
// ===== library: MasterCopy "Pallet dispenser" =====

FUNCTION_BLOCK "Pallet dispenser"   // FB4, LAD
{ S7_Optimized_Access := 'FALSE' }
VERSION : 0.1
   VAR_INPUT
      DOWN_accident : Bool;
      Dispenser_is_down : Bool;
      Dispenser_in_middle : Bool;
      Dispenser_is_up : Bool;
      UP_accident : Bool;
      Circuit_breaker : Bool;
      Arms_are_open : Bool;
      Arms_are_close : Bool;
      Pallet_under_dispenser : Bool;
      Automatic_mode : Bool;
      Power_circuit_OK : Bool;
      Pneumatic_OK : Bool;
      Sensor_before_dispenser : Bool;
      Button_Open_door : Bool;
      Sensor_door_are_open : Bool;
      Button_Door_are_close : Bool;
      OP_up : Bool;
      OP_down : Bool;
      OP_Airs_move : Bool;
      Pallet_transfare : Bool;
      Button_RESET : Bool;
   END_VAR
   VAR_OUTPUT
      Let_go_UP : Bool;
      Let_go_DOWN : Bool;
      Break : Bool;
      Let_arms_close : Bool;
      Let_arms_open : Bool;
      Let_open_door : Bool;
      Led_door_are_open : Bool;
   END_VAR
   VAR
      Paleta_polozena : Bool;
      Stop_v_rucnim : Bool;
      Hrana_stop_v_rucnim : Bool;
      Pozadavek_otevreni_dveri : Bool;
      Door_opened : Bool;
      Arms_are_close_pozition : Bool;
   END_VAR
   VAR_TEMP   // added for the SCL form of the ladder/FBD networks
      _s5time1 : S5Time;
      _w1 : Bool;
   END_VAR
BEGIN

REGION Network 1
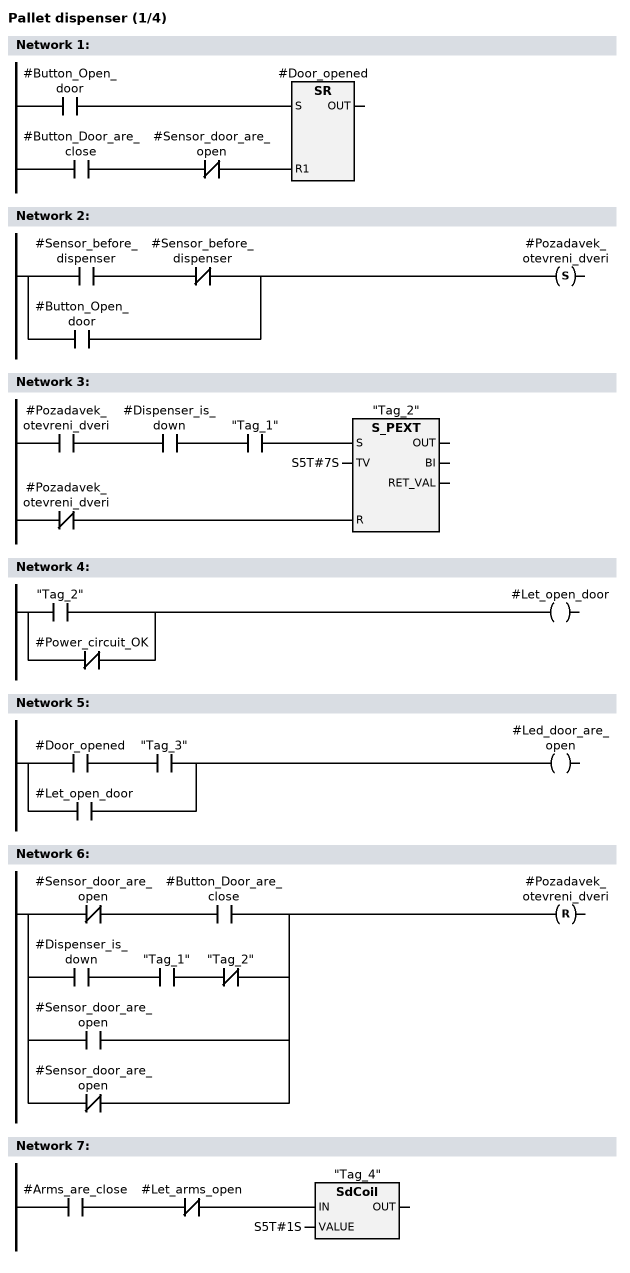
   IF #Button_Open_door THEN
       #Door_opened := TRUE;   // SR flip-flop
   END_IF;
   IF #Button_Door_are_close AND NOT #Sensor_door_are_open THEN #Door_opened := FALSE; END_IF;
END_REGION

REGION Network 2
   RUNG wire#powerrail
      Contact( #Sensor_before_dispenser )
      I_Contact( #Sensor_before_dispenser )
      wire#w1
      S_Coil( #Pozadavek_otevreni_dveri )
   END_RUNG
   RUNG wire#powerrail
      Contact( #Button_Open_door )
   END_RUNG wire#w1
   // the same network as SCL:
   IF (#Sensor_before_dispenser AND NOT #Sensor_before_dispenser) OR #Button_Open_door THEN
       #Pozadavek_otevreni_dveri := TRUE;
   END_IF;
END_REGION

REGION Network 3
   RUNG wire#powerrail
      Contact( #Pozadavek_otevreni_dveri )
      Contact( #Dispenser_is_down )
      Contact( "Tag_1" )
      S_PEXT(T_NO := "Tag_2", TV := S5T#7S, R := wire#w1, BI =>, RET_VAL =>)
   END_RUNG
   RUNG wire#powerrail
      I_Contact( #Pozadavek_otevreni_dveri )
   END_RUNG wire#w1
   // the same network as SCL:
   #_s5time1 := S_PEXT(T_NO := "Tag_2",
                       TV := S5T#7S,
                       S := #Pozadavek_otevreni_dveri AND #Dispenser_is_down AND "Tag_1",
                       R := NOT #Pozadavek_otevreni_dveri);
END_REGION

REGION Network 4
   RUNG wire#powerrail
      Contact( "Tag_2" )
      wire#w1
      Coil( #Let_open_door )
   END_RUNG
   RUNG wire#powerrail
      I_Contact( #Power_circuit_OK )
   END_RUNG wire#w1
   // the same network as SCL:
   #Let_open_door := "Tag_2" OR NOT #Power_circuit_OK;
END_REGION

REGION Network 5
   #Led_door_are_open := #Let_open_door OR (#Door_opened AND "Tag_3");
END_REGION

REGION Network 6
   RUNG wire#powerrail
      I_Contact( #Sensor_door_are_open )
      Contact( #Button_Door_are_close )
      wire#w1
      R_Coil( #Pozadavek_otevreni_dveri )
   END_RUNG
   RUNG wire#powerrail
      Contact( #Dispenser_is_down )
      Contact( "Tag_1" )
      I_Contact( "Tag_2" )
   END_RUNG wire#w1
   RUNG wire#powerrail
      Contact( #Sensor_door_are_open )
   END_RUNG wire#w1
   RUNG wire#powerrail
      I_Contact( #Sensor_door_are_open )
   END_RUNG wire#w1
   // the same network as SCL:
   IF (NOT #Sensor_door_are_open AND #Button_Door_are_close) OR (#Dispenser_is_down AND "Tag_1" AND NOT "Tag_2") OR #Sensor_door_are_open OR NOT #Sensor_door_are_open THEN
       #Pozadavek_otevreni_dveri := FALSE;
   END_IF;
END_REGION

REGION Network 7
   // no SCL statement known for SdCoil: written as a call
   SdCoil(value := S5T#1S, operand := "Tag_4", in := #Arms_are_close AND NOT #Let_arms_open);
END_REGION

REGION Network 8
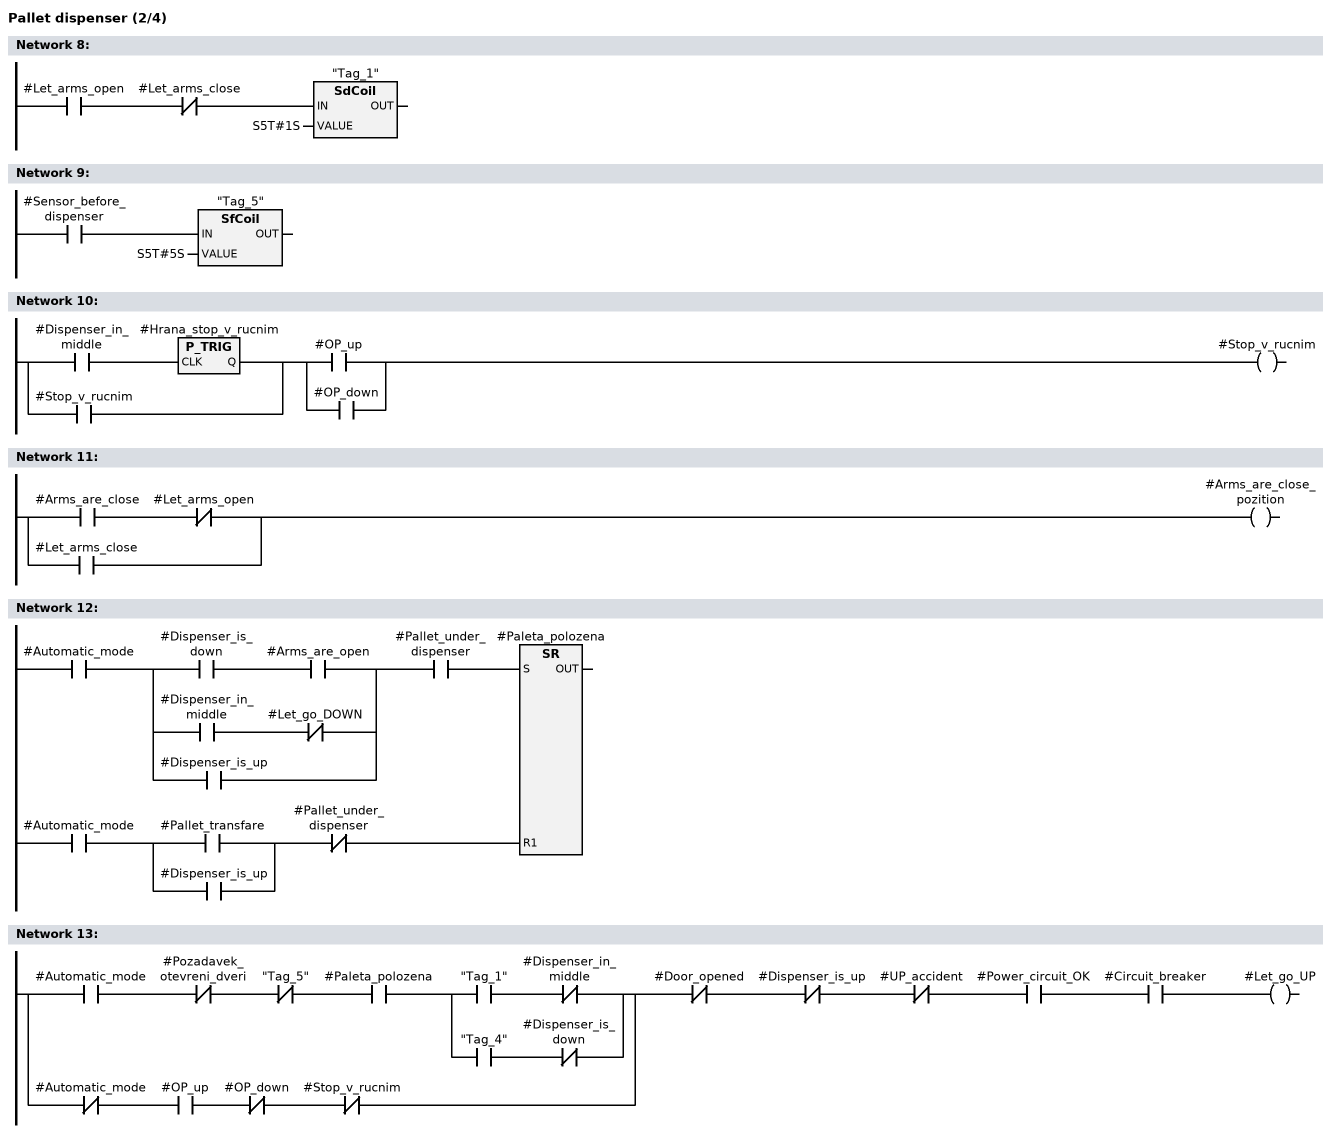
   // no SCL statement known for SdCoil: written as a call
   SdCoil(value := S5T#1S, operand := "Tag_1", in := #Let_arms_open AND NOT #Let_arms_close);
END_REGION

REGION Network 9
   // no SCL statement known for SfCoil: written as a call
   SfCoil(value := S5T#5S, operand := "Tag_5", in := #Sensor_before_dispenser);
END_REGION

REGION Network 10
   RUNG wire#powerrail
      Contact( #Dispenser_in_middle )
      P_Trig( #Hrana_stop_v_rucnim )
      wire#w1
      Contact( #OP_up )
      wire#w2
      Coil( #Stop_v_rucnim )
   END_RUNG
   RUNG wire#powerrail
      Contact( #Stop_v_rucnim )
   END_RUNG wire#w1
   RUNG wire#w1
      Contact( #OP_down )
   END_RUNG wire#w2
   // the same network as SCL:
   #_w1 := #Dispenser_in_middle AND NOT #Hrana_stop_v_rucnim;   // rising edge
   #Hrana_stop_v_rucnim := #Dispenser_in_middle;
   #Stop_v_rucnim := (#_w1 OR #Stop_v_rucnim) AND (#OP_up OR #OP_down);
END_REGION

REGION Network 11
   RUNG wire#powerrail
      Contact( #Arms_are_close )
      I_Contact( #Let_arms_open )
      wire#w1
      Coil( #Arms_are_close_pozition )
   END_RUNG
   RUNG wire#powerrail
      Contact( #Let_arms_close )
   END_RUNG wire#w1
   // the same network as SCL:
   #Arms_are_close_pozition := (#Arms_are_close AND NOT #Let_arms_open) OR #Let_arms_close;
END_REGION

REGION Network 12
   IF #Automatic_mode AND ((#Dispenser_is_down AND #Arms_are_open) OR (#Dispenser_in_middle AND NOT #Let_go_DOWN) OR #Dispenser_is_up) AND #Pallet_under_dispenser THEN
       #Paleta_polozena := TRUE;   // SR flip-flop
   END_IF;
   IF #Automatic_mode AND (#Pallet_transfare OR #Dispenser_is_up) AND NOT #Pallet_under_dispenser THEN
       #Paleta_polozena := FALSE;
   END_IF;
END_REGION

REGION Network 13
   #Let_go_UP := ((#Automatic_mode AND NOT #Pozadavek_otevreni_dveri AND NOT "Tag_5" AND #Paleta_polozena AND (("Tag_1" AND NOT #Dispenser_in_middle) OR ("Tag_4" AND NOT #Dispenser_is_down))) OR (NOT #Automatic_mode AND #OP_up AND NOT #OP_down AND NOT #Stop_v_rucnim)) AND NOT #Door_opened AND NOT #Dispenser_is_up AND NOT #UP_accident AND #Power_circuit_OK AND #Circuit_breaker;
END_REGION

REGION Network 14
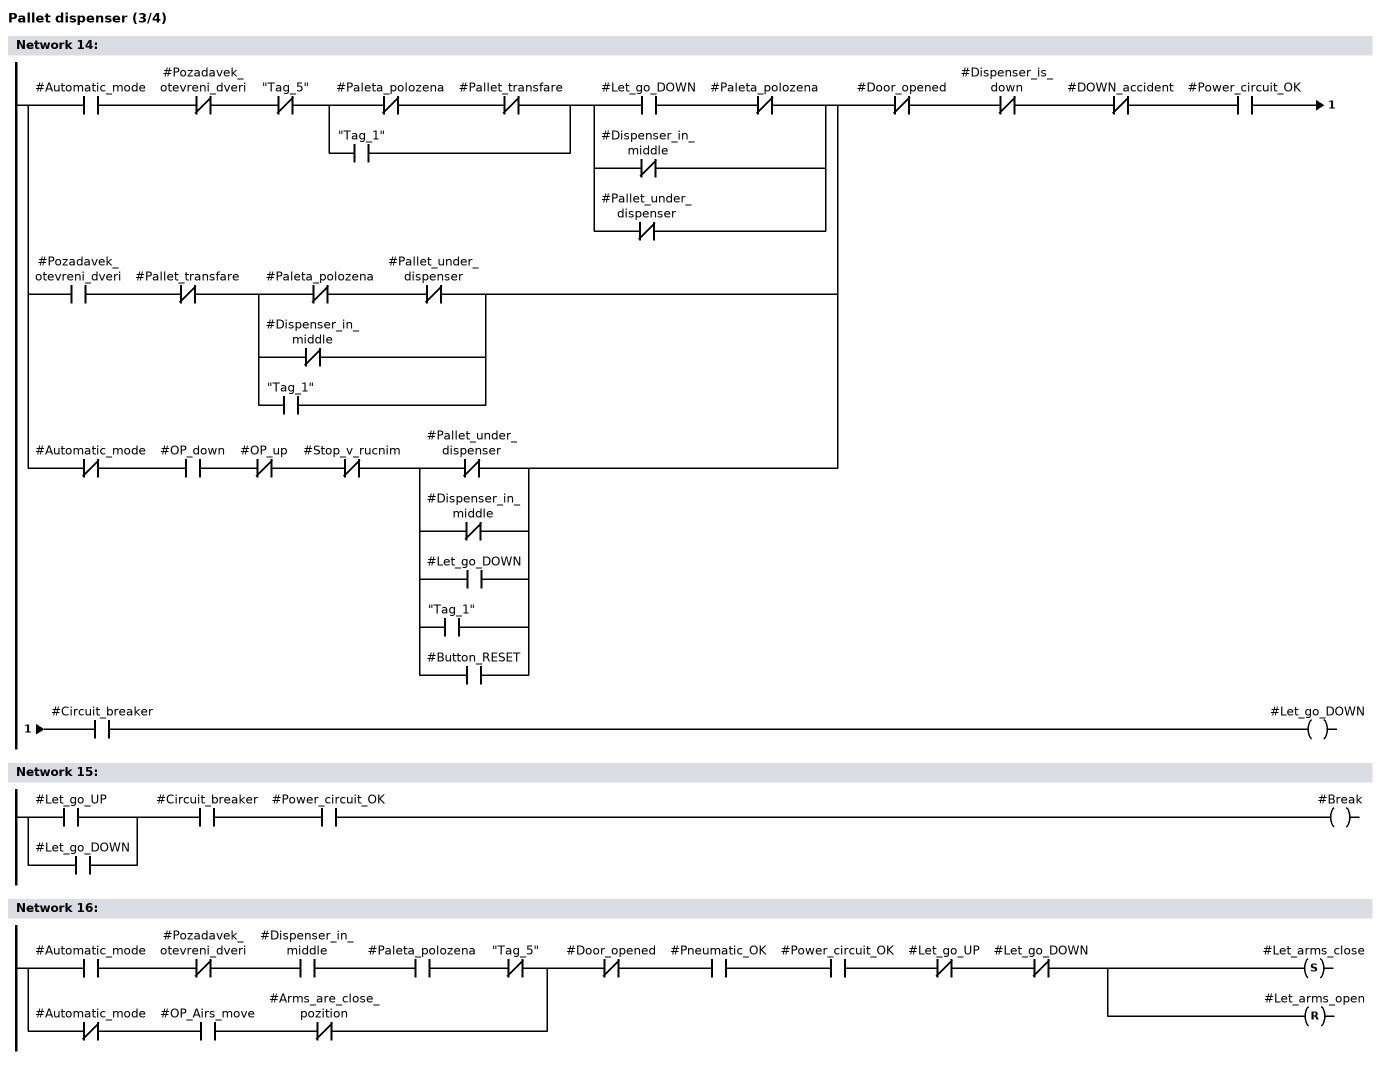
   #Let_go_DOWN := ((#Automatic_mode AND NOT #Pozadavek_otevreni_dveri AND NOT "Tag_5" AND ((NOT #Paleta_polozena AND NOT #Pallet_transfare) OR "Tag_1") AND (NOT #Dispenser_in_middle OR NOT #Pallet_under_dispenser OR (#Let_go_DOWN AND NOT #Paleta_polozena))) OR (#Pozadavek_otevreni_dveri AND NOT #Pallet_transfare AND (NOT #Dispenser_in_middle OR (NOT #Paleta_polozena AND NOT #Pallet_under_dispenser) OR "Tag_1")) OR (NOT #Automatic_mode AND #OP_down AND NOT #OP_up AND NOT #Stop_v_rucnim AND (NOT #Pallet_under_dispenser OR NOT #Dispenser_in_middle OR #Let_go_DOWN OR "Tag_1" OR #Button_RESET))) AND NOT #Door_opened AND NOT #Dispenser_is_down AND NOT #DOWN_accident AND #Power_circuit_OK AND #Circuit_breaker;
END_REGION

REGION Network 15
   RUNG wire#powerrail
      Contact( #Let_go_UP )
      wire#w1
      Contact( #Circuit_breaker )
      Contact( #Power_circuit_OK )
      Coil( #Break )
   END_RUNG
   RUNG wire#powerrail
      Contact( #Let_go_DOWN )
   END_RUNG wire#w1
   // the same network as SCL:
   #Break := (#Let_go_UP OR #Let_go_DOWN) AND #Circuit_breaker AND #Power_circuit_OK;
END_REGION

REGION Network 16
   RUNG wire#powerrail
      Contact( #Automatic_mode )
      I_Contact( #Pozadavek_otevreni_dveri )
      Contact( #Dispenser_in_middle )
      Contact( #Paleta_polozena )
      I_Contact( "Tag_5" )
      wire#w1
      I_Contact( #Door_opened )
      Contact( #Pneumatic_OK )
      Contact( #Power_circuit_OK )
      I_Contact( #Let_go_UP )
      I_Contact( #Let_go_DOWN )
      wire#w2
      S_Coil( #Let_arms_close )
   END_RUNG
   RUNG wire#powerrail
      I_Contact( #Automatic_mode )
      Contact( #OP_Airs_move )
      I_Contact( #Arms_are_close_pozition )
   END_RUNG wire#w1
   RUNG wire#w2
      R_Coil( #Let_arms_open )
   END_RUNG
   // the same network as SCL:
   IF ((#Automatic_mode AND NOT #Pozadavek_otevreni_dveri AND #Dispenser_in_middle AND #Paleta_polozena AND NOT "Tag_5") OR (NOT #Automatic_mode AND #OP_Airs_move AND NOT #Arms_are_close_pozition)) AND NOT #Door_opened AND #Pneumatic_OK AND #Power_circuit_OK AND NOT #Let_go_UP AND NOT #Let_go_DOWN THEN
       #Let_arms_close := TRUE;
       #Let_arms_open := FALSE;
   END_IF;
END_REGION

REGION Network 17
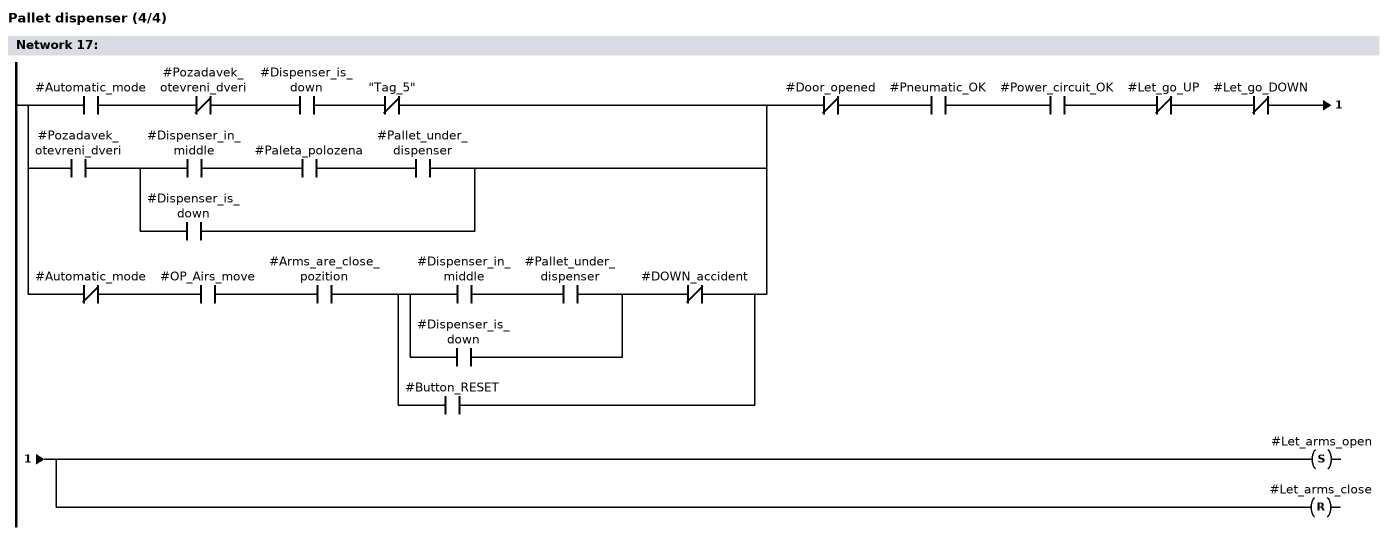
   IF ((#Automatic_mode AND NOT #Pozadavek_otevreni_dveri AND #Dispenser_is_down AND NOT "Tag_5") OR (#Pozadavek_otevreni_dveri AND ((#Dispenser_in_middle AND #Paleta_polozena AND #Pallet_under_dispenser) OR #Dispenser_is_down)) OR (NOT #Automatic_mode AND #OP_Airs_move AND #Arms_are_close_pozition AND (((#Dispenser_is_down OR (#Dispenser_in_middle AND #Pallet_under_dispenser)) AND NOT #DOWN_accident) OR #Button_RESET))) AND NOT #Door_opened AND #Pneumatic_OK AND #Power_circuit_OK AND NOT #Let_go_UP AND NOT #Let_go_DOWN THEN
       #Let_arms_open := TRUE;
       #Let_arms_close := FALSE;
   END_IF;
END_REGION
END_FUNCTION_BLOCK